FUNCTION_BLOCK Seq_Set_Plate_2 EXTENDS FB_Basis IMPLEMENTS I_Sequenz
VAR_INPUT
	// Skillzuweisung
	R_Move			:I_Skill_RoboterErweitert;
	G_Move			:I_Skill_SmartGreifer; 
	
	// Prozessparameter		
	RobParam				:ARRAY[0..3] OF sRoboterProzessVariablen;
	GripParam				:sSmartGreiferProzessVariablen;
	ErreichtParam			:sKraftVariablen;
END_VAR
VAR_OUTPUT
	
END_VAR
VAR
	
END_VAR

// Ablauf
ACT_Ablauf();

// Zustandshandling
CASE iState OF
	0:	// BEREIT
		IF bStart THEN
			iState := 1;
		END_IF
	1:	// LAUFEND
		IF eSysCommand = 4 THEN
			bReset := TRUE;
			SFCReset := TRUE;
		END_IF
		
		IF bBeendet OR bReset THEN
			bReset := FALSE;
			SFCReset := FALSE;
			iState := 0;
		END_IF
	2: // ABGESCHLOSSEN
		IF SFCCurrentStep = 'Init' THEN
			iState := 0;
		END_IF
END_CASE

ACTION ACT_Ablauf:
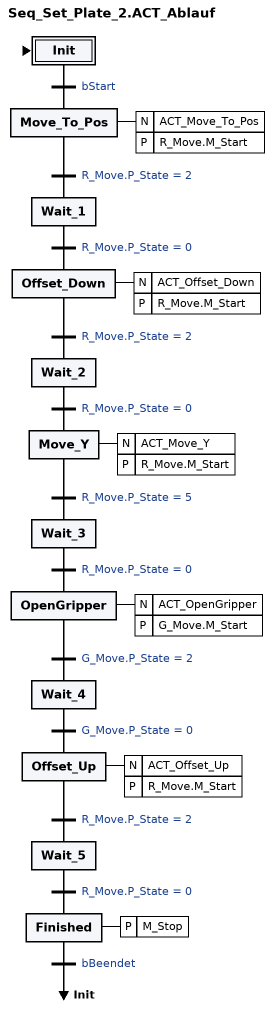
INITIAL_STEP Init:
END_STEP
TRANSITION FROM Init TO Move_To_Pos
    := bStart;
END_TRANSITION
STEP Move_To_Pos:
    ACT_Move_To_Pos(N);
    R_Move.M_Start(P);
END_STEP
TRANSITION FROM Move_To_Pos TO Wait_1
    := R_Move.P_State = 2;
END_TRANSITION
STEP Wait_1:
END_STEP
TRANSITION FROM Wait_1 TO Offset_Down
    := R_Move.P_State = 0;
END_TRANSITION
STEP Offset_Down:
    ACT_Offset_Down(N);
    R_Move.M_Start(P);
END_STEP
TRANSITION FROM Offset_Down TO Wait_2
    := R_Move.P_State = 2;
END_TRANSITION
STEP Wait_2:
END_STEP
TRANSITION FROM Wait_2 TO Move_Y
    := R_Move.P_State = 0;
END_TRANSITION
STEP Move_Y:
    ACT_Move_Y(N);
    R_Move.M_Start(P);
END_STEP
TRANSITION FROM Move_Y TO Wait_3
    := R_Move.P_State = 5;
END_TRANSITION
STEP Wait_3:
END_STEP
TRANSITION FROM Wait_3 TO OpenGripper
    := R_Move.P_State = 0;
END_TRANSITION
STEP OpenGripper:
    ACT_OpenGripper(N);
    G_Move.M_Start(P);
END_STEP
TRANSITION FROM OpenGripper TO Wait_4
    := G_Move.P_State = 2;
END_TRANSITION
STEP Wait_4:
END_STEP
TRANSITION FROM Wait_4 TO Offset_Up
    := G_Move.P_State = 0;
END_TRANSITION
STEP Offset_Up:
    ACT_Offset_Up(N);
    R_Move.M_Start(P);
END_STEP
TRANSITION FROM Offset_Up TO Wait_5
    := R_Move.P_State = 2;
END_TRANSITION
STEP Wait_5:
END_STEP
TRANSITION FROM Wait_5 TO Finished
    := R_Move.P_State = 0;
END_TRANSITION
STEP Finished:
    M_Stop(P);
END_STEP
TRANSITION FROM Finished TO Init
    := bBeendet;
END_TRANSITION
END_ACTION

ACTION ACT_Move_To_Pos:
R_Move.P_RobotParam := RobParam[0];
END_ACTION

ACTION ACT_Move_Y:
R_Move.P_RobotParam := RobParam[2];
R_Move.P_Erreicht := ErreichtParam;
END_ACTION

ACTION ACT_Offset_Down:
R_Move.P_RobotParam := RobParam[1];
END_ACTION

ACTION ACT_Offset_Up:
R_Move.P_RobotParam := RobParam[3];
END_ACTION

ACTION ACT_OpenGripper:
G_Move.P_SGripperParam := GripParam;
END_ACTION

END_FUNCTION_BLOCK

(* stored: Version 1.1.0.1
   POU Seq_Set_Plate_2: Id {a043f3d5-8415-4a96-8d41-cb1dde8c9015}, SpecialFunc None
   Folder 01_Zuweisung: Id {4391b0a4-0c91-4829-a6cc-8809298300f2}
   Action ACT_Ablauf: Id {6f5e0941-b13a-4ff9-bd21-2874ddc8bf8a}
   Action ACT_Move_To_Pos: Id {78bb210d-b6fe-44a8-ac2e-3e4589e08090}
   Action ACT_Move_Y: Id {3cd6a614-878a-4ed2-9388-c85b709feeed}
   Action ACT_Offset_Down: Id {d1b14132-3d57-410a-8335-7c4792bcc75e}
   Action ACT_Offset_Up: Id {d243429e-097b-4af0-8ef0-9acfc886aa83}
   Action ACT_OpenGripper: Id {ba7bd6bb-a5eb-4fb1-9501-0a15a5c3587b} *)
